FUNCTION_BLOCK FB_ProfidriveTelegram1_Test EXTENDS TcUnit.FB_TestSuite

Test_ProcessDataControl();
Test_ProcessDataStatus();
Test_Cycle_Status_Const_Mirror();

METHOD Test_Cycle_Status_Const_Mirror : REFERENCE TO FB_Test
VAR
	fbDrive 			: FB_Profidrive_Telegram1;
	bExpected			: BOOL;
	stExpected			: ST_Profidrive_Telegram1_Status;
	bResult 			: BOOL;	
	stResult			: ST_Profidrive_Telegram1_Status;
	
	stSetControl		: ST_Profidrive_Telegram1_Control;
END_VAR
TEST('Status CONST TRUE');

bExpected := TRUE;

fbDrive.Cycle();

stResult := fbDrive.stStatus;

bResult := BIT_TO_BOOL(stResult.b8_DeviationWithinTolerance);

AssertEquals(Expected := bExpected,
             Actual := bResult,
             Message := 'DeviationWithinTolerance not set correctly');

bResult := BIT_TO_BOOL(stResult.b11_TorqueOrPowerLimitNotReached);
			 
AssertEquals(Expected := bExpected,
             Actual := bResult,
             Message := 'TorqueOrPowerLimitNotReached not set correctly');
			 
bResult := BIT_TO_BOOL(stResult.b13_NoOvertempAlarm);
			 
AssertEquals(Expected := bExpected,
             Actual := bResult,
             Message := 'NoOvertempAlarm not set correctly');

bResult := BIT_TO_BOOL(stResult.b15_NoAlarmNoOvertempPowerUnit);
			 
AssertEquals(Expected := bExpected,
             Actual := bResult,
             Message := 'NoAlarmNoOvertempPowerUnit not set correctly');
	 
TEST_FINISHED();

TEST('Status CONST FALSE');

bExpected := FALSE;

fbDrive.Cycle();

stResult := fbDrive.stStatus;

bResult := BIT_TO_BOOL(stResult.b3_FaultPresent);

AssertEquals(Expected := bExpected,
             Actual := bResult,
             Message := 'FaultPresent not set correctly');

bResult := BIT_TO_BOOL(stResult.b7_AlarmPresent);
			 
AssertEquals(Expected := bExpected,
             Actual := bResult,
             Message := 'AlarmPresent not set correctly');
TEST_FINISHED();

TEST('Status Mirror Control FALSE');

bExpected := FALSE;

stSetControl.b3_EnableOperation := bExpected;

fbDrive.stConfig.bControlRequested := bExpected;

fbDrive.stControl := stSetControl;

fbDrive.Cycle();

stResult := fbDrive.stStatus;

bResult := BIT_TO_BOOL(stResult.b2_OperationEnabled);
			 
AssertEquals(Expected := bExpected,
             Actual := bResult,
             Message := 'OperationEnabled not set correctly');

bResult := BIT_TO_BOOL(stResult.b9_ControlRequested);
			 
AssertEquals(Expected := bExpected,
             Actual := bResult,
             Message := 'ControlRequested not set correctly');

TEST_FINISHED();

TEST('Status Mirror Control TRUE');

bExpected := TRUE;

stSetControl.b3_EnableOperation := bExpected;

fbDrive.stConfig.bControlRequested := bExpected;

fbDrive.stControl := stSetControl;

fbDrive.Cycle();

stResult := fbDrive.stStatus;

bResult := BIT_TO_BOOL(stResult.b2_OperationEnabled);
			 
AssertEquals(Expected := bExpected,
             Actual := bResult,
             Message := 'OperationEnabled not set correctly');

bResult := BIT_TO_BOOL(stResult.b9_ControlRequested);
			 
AssertEquals(Expected := bExpected,
             Actual := bResult,
             Message := 'ControlRequested not set correctly');
	 
TEST_FINISHED();
END_METHOD

METHOD Test_ProcessDataControl : REFERENCE TO FB_Test
VAR
	fbDrive 					: FB_Profidrive_Telegram1;
	
	nExpectedSTW1 				: WORD;
	nExpectedTargetVelocity 	: INT;
	nActualSTW1 				: WORD;
	nActualTargetVelocity		: INT;	
		
	aExpectedControlData 		: ST_Profidrive_Telegram1_Control;		
	aActualControlData			: ST_Profidrive_Telegram1_Control;	
END_VAR
TEST('Process data to control structure');

//Arrange
nExpectedSTW1 := 16#A1B2;
nExpectedTargetVelocity := UINT_TO_INT(16#C3D4);

F_Memcpy(ADR(aExpectedControlData), ADR(nExpectedSTW1), 2, FALSE);
F_Memcpy(ADR(aExpectedControlData) + 2, ADR(nExpectedTargetVelocity), 2, FALSE);

fbDrive.pControl := ADR(aExpectedControlData);

//Act
fbDrive.GetControlData();

//Assert
F_Memcpy(ADR(nActualSTW1), ADR(fbDrive.stControl), 2, FALSE);
F_Memcpy(ADR(nActualTargetVelocity), ADR(fbDrive.stControl) + 2, 2, FALSE);

AssertEquals(Expected := nExpectedSTW1,
             Actual := nActualSTW1,
             Message := 'STW1 is not correct');
	 
AssertEquals(Expected := nExpectedTargetVelocity,
             Actual := nActualTargetVelocity,
             Message := 'TargetVelocity is not correct');

TEST_FINISHED();


TEST('Process data to control structure SWAP');

//Arrange
nExpectedSTW1 := 16#C3F3;
nExpectedTargetVelocity := UINT_TO_INT(16#C3F3);

F_Memcpy(ADR(aExpectedControlData), ADR(nExpectedSTW1), 2, TRUE);
F_Memcpy(ADR(aExpectedControlData) + 2, ADR(nExpectedTargetVelocity), 2, TRUE);

fbDrive.stConfig.bSwapProcessData := TRUE;

fbDrive.pControl := ADR(aExpectedControlData);

//Act
fbDrive.GetControlData();

//Assert
F_Memcpy(ADR(nActualSTW1), ADR(fbDrive.stControl), 2, FALSE);
F_Memcpy(ADR(nActualTargetVelocity), ADR(fbDrive.stControl) + 2, 2, FALSE);

AssertEquals(Expected := nExpectedSTW1,
             Actual := nActualSTW1,
             Message := 'STW1 is not correct');
	 
AssertEquals(Expected := nExpectedTargetVelocity,
             Actual := nActualTargetVelocity,
             Message := 'TargetVelocity is not correct');	

TEST_FINISHED();
END_METHOD

METHOD Test_ProcessDataStatus : REFERENCE TO FB_Test
VAR
	fbDrive 					: FB_Profidrive_Telegram1;
	
	nExpectedZSW1 				: WORD;
	nExpectedActualVelocity		: INT;	
	nActualZSW1 				: WORD;
	nActualActualVelocity		: INT;	

	stExpectedStatusData 		: ST_Profidrive_Telegram1_Status;		
	stActualStatusData 			: ST_Profidrive_Telegram1_Status;	
END_VAR
TEST('Assign status structure to process data');

//Arrange
nExpectedZSW1 := 16#A1B2;
nExpectedActualVelocity := UINT_TO_INT(16#C3D4);
F_Memcpy(ADR(fbDrive.stStatus), ADR(nExpectedZSW1), 2, FALSE);
F_Memcpy(ADR(fbDrive.stStatus) + 2, ADR(nExpectedActualVelocity), 2, FALSE);

fbDrive.pStatus := ADR(stActualStatusData);

//Act
fbDrive.SetStatusData();

//Assert
F_Memcpy(ADR(nActualZSW1), ADR(stActualStatusData), 2, FALSE);
F_Memcpy(ADR(nActualActualVelocity), ADR(stActualStatusData) + 2, 2, FALSE);

AssertEquals(Expected := nExpectedZSW1,
             Actual := nActualZSW1,
             Message := 'ZSW1 is not correct');
	 
AssertEquals(Expected := nExpectedActualVelocity,
             Actual := nActualActualVelocity,
             Message := 'ActualVelocity is not correct');	

TEST_FINISHED();


TEST('Assign status structure to process data SWAP');

//Arrange
nExpectedZSW1 := 16#A1B2;
nExpectedActualVelocity	:= UINT_TO_INT(16#C3D4);

F_Memcpy(ADR(fbDrive.stStatus), ADR(nExpectedZSW1), 2, FALSE);
F_Memcpy(ADR(fbDrive.stStatus) + 2, ADR(nExpectedActualVelocity), 2, FALSE);

fbDrive.stConfig.bSwapProcessData := TRUE;
fbDrive.pStatus := ADR(stActualStatusData);

//Act
fbDrive.SetStatusData();

//Assert
F_Memcpy(ADR(nActualZSW1), ADR(stActualStatusData), 2, TRUE);
F_Memcpy(ADR(nActualActualVelocity), ADR(stActualStatusData) + 2, 2, TRUE);

AssertEquals(Expected := nExpectedZSW1,
             Actual := nActualZSW1,
             Message := 'ZSW1 is not correct');
	 
AssertEquals(Expected := nExpectedActualVelocity,
             Actual := nActualActualVelocity,
             Message := 'ActualVelocity is not correct');	

TEST_FINISHED();
END_METHOD

END_FUNCTION_BLOCK

(* stored: Version 1.1.0.1, ProductVersion 3.1.4024.12
   POU FB_ProfidriveTelegram1_Test: Id {a3b4595a-ff1b-0df3-298e-dfe9bd1cbb12}, SpecialFunc None
   Method Test_Cycle_Status_Const_Mirror: Id {db390c1c-177c-056e-14f1-4fd968bd1454}
   Method Test_ProcessDataControl: Id {16ebd94e-bdad-08df-3f30-2d8391d4539e}
   Method Test_ProcessDataStatus: Id {4abedd89-dcb3-0b8f-04ba-e93a9c2d32c9} *)
